// TIA Portal V19 export
TYPE "LEXCHANGETRAY_typeConstraintRollerEm_toRollerDeliver"
// stored: Access Published
   STRUCT
      feedback : "LEXCHANGETRAY_typeConstraintRollerEm_toRollerFeedback";
      req : "LEXCHANGETRAY_typeConstraintRollerEm_toRollerReq";
   END_STRUCT;
END_TYPE
